// TIA Portal V20 export
// export: Created 2026-10-01T22:10:06.1398792Z, ExportSetting WithDefaults, DisplayName Totally Integrated Automation Portal, DisplayVersion V20, DisplayName TIA Portal Openness, DisplayVersion V20, DisplayName TIA Portal Version Control Interface, DisplayVersion V20, DisplayName SINAMICS Startdrive Advanced, DisplayVersion V20, DisplayName SINAMICS Startdrive G130, G150, S120, S150, SINAMICS MV, G220, S200, S210, DisplayVersion V20, DisplayName SINAMICS Startdrive G110M, G120, G120C, G120D, G120P, G115D, DisplayVersion V20, DisplayName STEP 7 Professional, DisplayVersion V20, DisplayName STEP 7 Safety, DisplayVersion V20, DisplayName WinCC Basic/Comfort/Advanced, DisplayVersion V20, DisplayName WinCC Unified, DisplayVersion V20
FUNCTION_BLOCK "ZZ_LadTest_Mul"   // FB26, LAD
{ S7_Optimized_Access := 'TRUE' }
VERSION : 0.1
// stored: AutoNumber true, IsIECCheckEnabled false, IsRetainMemResEnabled false, MemoryReserve 100, SetENOAutomatically false, UDAEnableTagReadback false
   VAR_INPUT
      Start : Bool;
      "A" : Int;
      "B" : Int;
      X : Real;
   END_VAR
   VAR
      R1 : Int;
      R2 : Int;
      R3 : Int;
      R4 : Int;
      R5 : Int;
      Nrm : Real;
      Scl : Real;
      Latch : Bool;
      Latch2 : Bool;
   END_VAR
BEGIN

REGION Network 1
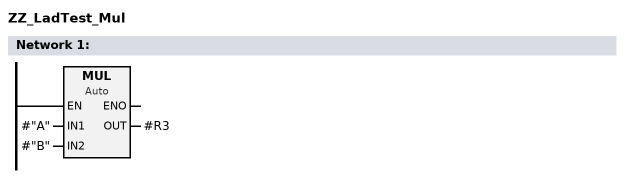
   RUNG wire#powerrail
      Mul(in1 := #"A", in2 := #"B", out => #R3)
   END_RUNG
   // the same network as SCL:
   #R3 := #"A" * #"B";
END_REGION
END_FUNCTION_BLOCK
